(* Timers. Hold DelayPB TRUE for 3 s and DelayLamp lights (watch DelayET count). Turn FanSwitch TRUE then FALSE: Fan runs on for 5 s. *)

PROGRAM P2_Timers
  VAR
    DelayPB : BOOL; (* Push-button that must be held for 3 s *)
    DelayLamp : BOOL; (* Lights after DelayPB has been held for 3 s *)
    DelayTimer : TON; (* On-delay timer instance *)
    DelayET : TIME; (* Elapsed time of DelayTimer *)
    FanSwitch : BOOL; (* Fan on/off switch *)
    Fan : BOOL; (* Fan motor: keeps running 5 s after FanSwitch goes off *)
    RunOnTimer : TOF; (* Off-delay timer instance *)
    RunOnET : TIME; (* Elapsed time of RunOnTimer *)
  END_VAR

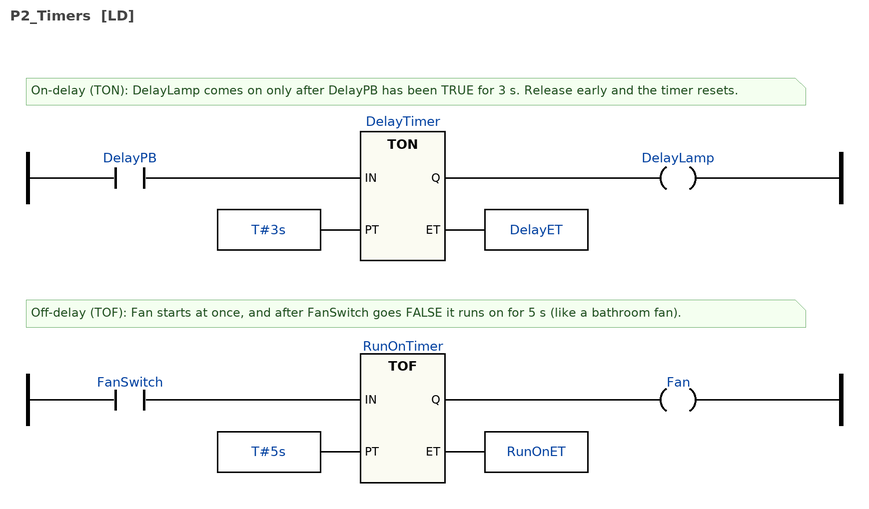
(* LD diagram, written out as Structured Text *)
(* On-delay (TON): DelayLamp comes on only after DelayPB has been TRUE for 3 s. Release early and the timer resets. *)
DelayTimer(IN := DelayPB, PT := T#3s);
DelayLamp := DelayTimer.Q;
DelayET := DelayTimer.ET;
(* Off-delay (TOF): Fan starts at once, and after FanSwitch goes FALSE it runs on for 5 s (like a bathroom fan). *)
RunOnTimer(IN := FanSwitch, PT := T#5s);
Fan := RunOnTimer.Q;
RunOnET := RunOnTimer.ET;
END_PROGRAM
